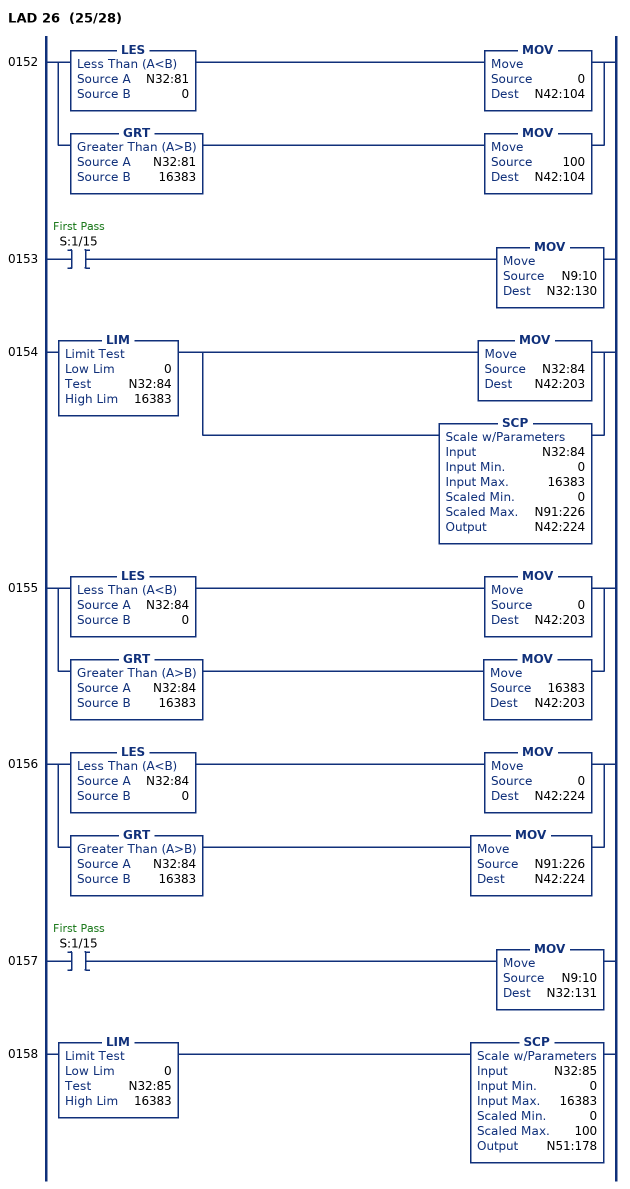
% Rung: 152 %
SOR BST LES N32:81 0 MOV 0 N42:104 NXB GRT N32:81 16383 MOV 100 N42:104 BND EOR
% Rung: 153 %
SOR XIC S:1/15 MOV N9:10 N32:130 EOR
%   S:1/15  "First Pass" %
% Rung: 154 %
SOR LIM 0 N32:84 16383 BST MOV N32:84 N42:203 NXB SCP N32:84 0 16383 0 N91:226 N42:224 BND EOR
% Rung: 155 %
SOR BST LES N32:84 0 MOV 0 N42:203 NXB GRT N32:84 16383 MOV 16383 N42:203 BND EOR
% Rung: 156 %
SOR BST LES N32:84 0 MOV 0 N42:224 NXB GRT N32:84 16383 MOV N91:226 N42:224 BND EOR
% Rung: 157 %
SOR XIC S:1/15 MOV N9:10 N32:131 EOR
%   S:1/15  "First Pass" %
% Rung: 158 %
SOR LIM 0 N32:85 16383 SCP N32:85 0 16383 0 100 N51:178 EOR

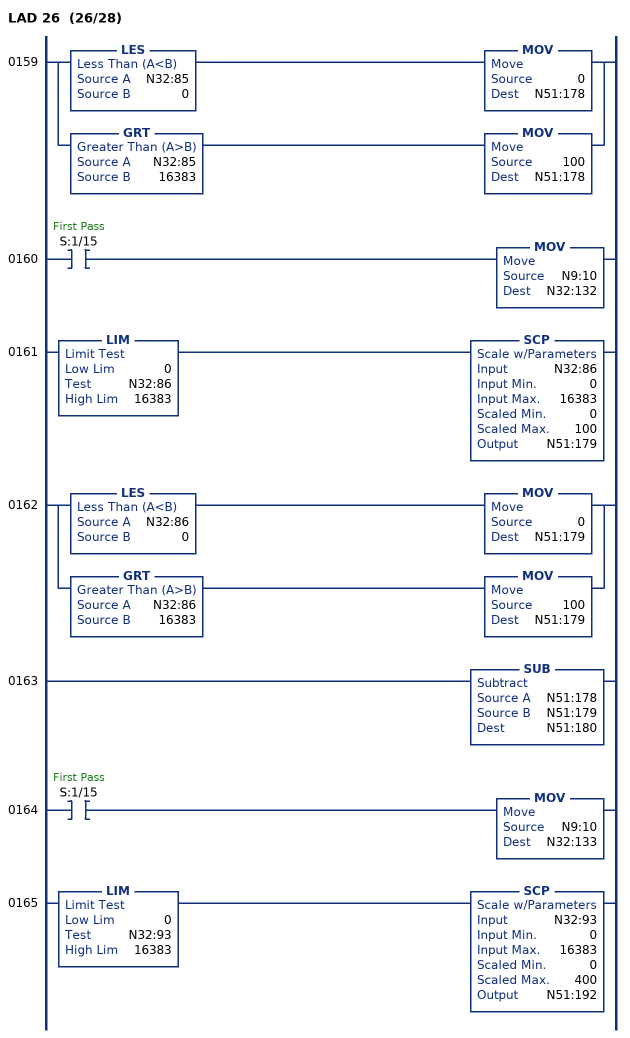
% Rung: 159 %
SOR BST LES N32:85 0 MOV 0 N51:178 NXB GRT N32:85 16383 MOV 100 N51:178 BND EOR
% Rung: 160 %
SOR XIC S:1/15 MOV N9:10 N32:132 EOR
%   S:1/15  "First Pass" %
% Rung: 161 %
SOR LIM 0 N32:86 16383 SCP N32:86 0 16383 0 100 N51:179 EOR
% Rung: 162 %
SOR BST LES N32:86 0 MOV 0 N51:179 NXB GRT N32:86 16383 MOV 100 N51:179 BND EOR
% Rung: 163 %
SOR SUB N51:178 N51:179 N51:180 EOR
% Rung: 164 %
SOR XIC S:1/15 MOV N9:10 N32:133 EOR
%   S:1/15  "First Pass" %
% Rung: 165 %
SOR LIM 0 N32:93 16383 SCP N32:93 0 16383 0 400 N51:192 EOR

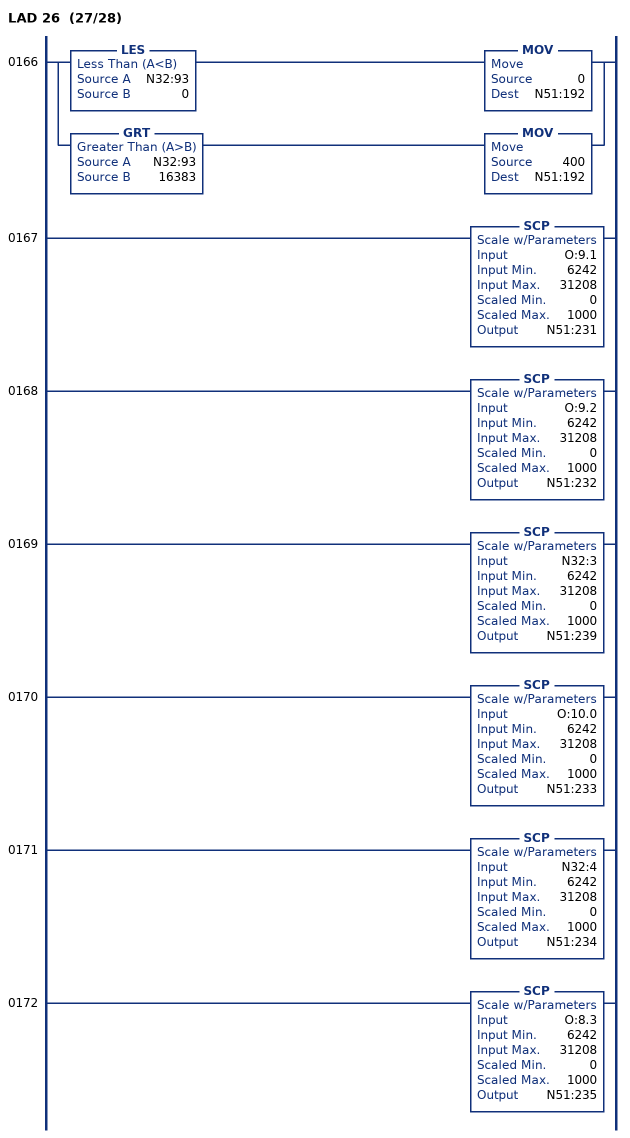
% Rung: 166 %
SOR BST LES N32:93 0 MOV 0 N51:192 NXB GRT N32:93 16383 MOV 400 N51:192 BND EOR
% Rung: 167 %
SOR SCP O:9.1 6242 31208 0 1000 N51:231 EOR
% Rung: 168 %
SOR SCP O:9.2 6242 31208 0 1000 N51:232 EOR
% Rung: 169 %
SOR SCP N32:3 6242 31208 0 1000 N51:239 EOR
% Rung: 170 %
SOR SCP O:10.0 6242 31208 0 1000 N51:233 EOR
% Rung: 171 %
SOR SCP N32:4 6242 31208 0 1000 N51:234 EOR
% Rung: 172 %
SOR SCP O:8.3 6242 31208 0 1000 N51:235 EOR

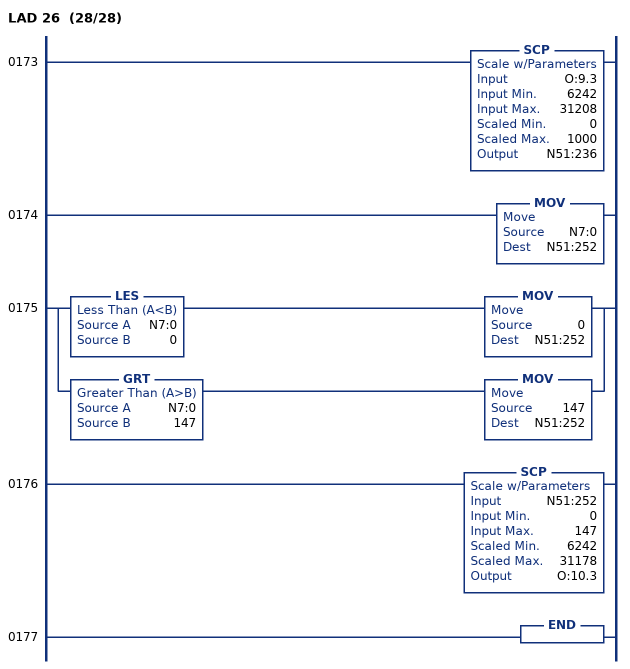
% Rung: 173 %
SOR SCP O:9.3 6242 31208 0 1000 N51:236 EOR
% Rung: 174 %
SOR MOV N7:0 N51:252 EOR
% Rung: 175 %
SOR BST LES N7:0 0 MOV 0 N51:252 NXB GRT N7:0 147 MOV 147 N51:252 BND EOR
% Rung: 176 %
SOR SCP N51:252 0 147 6242 31178 O:10.3 EOR
% Rung: 177 %
SOR END EOR

LADDER 27
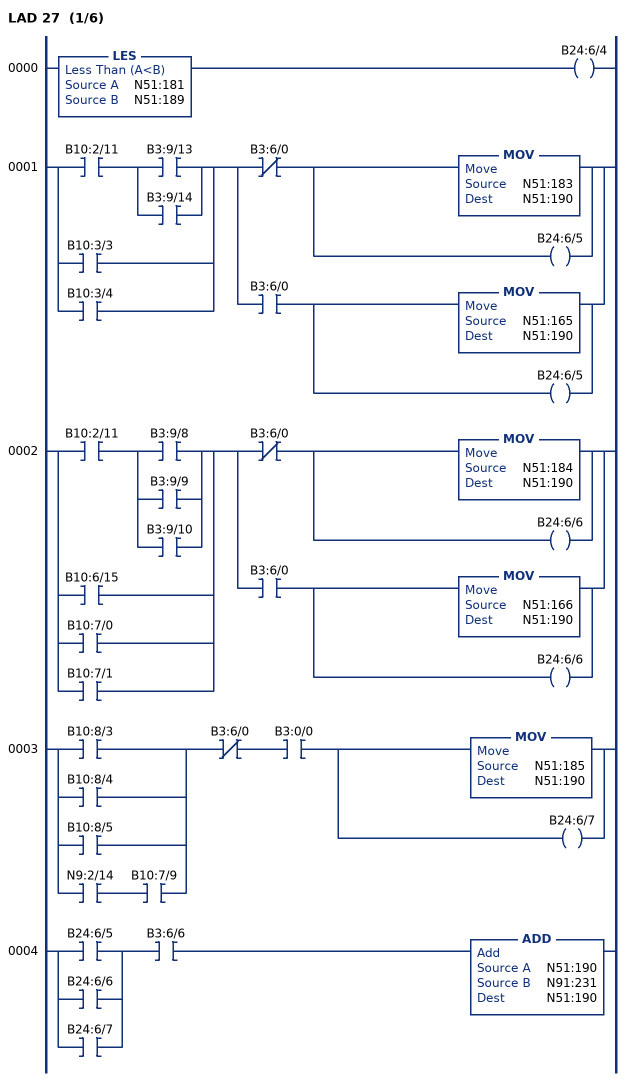
% Rung: 0 %
SOR LES N51:181 N51:189 OTE B24:6/4 EOR
% Rung: 1 %
SOR BST XIC B10:2/11 BST XIC B3:9/13 NXB XIC B3:9/14 BND NXB XIC B10:3/3 NXB XIC B10:3/4 BND BST XIO B3:6/0 BST MOV N51:183 N51:190 NXB OTE B24:6/5 BND NXB XIC B3:6/0 BST MOV N51:165 N51:190 NXB OTE B24:6/5 BND BND EOR
% Rung: 2 %
SOR BST XIC B10:2/11 BST XIC B3:9/8 NXB XIC B3:9/9 NXB XIC B3:9/10 BND NXB XIC B10:6/15 NXB XIC B10:7/0 NXB XIC B10:7/1 BND BST XIO B3:6/0 BST MOV N51:184 N51:190 NXB OTE B24:6/6 BND NXB XIC B3:6/0 BST MOV N51:166 N51:190 NXB OTE B24:6/6 BND BND EOR
% Rung: 3 %
SOR BST XIC B10:8/3 NXB XIC B10:8/4 NXB XIC B10:8/5 NXB XIC N9:2/14 XIC B10:7/9 BND XIO B3:6/0 XIC B3:0/0 BST MOV N51:185 N51:190 NXB OTE B24:6/7 BND EOR
% Rung: 4 %
SOR BST XIC B24:6/5 NXB XIC B24:6/6 NXB XIC B24:6/7 BND XIC B3:6/6 ADD N51:190 N91:231 N51:190 EOR

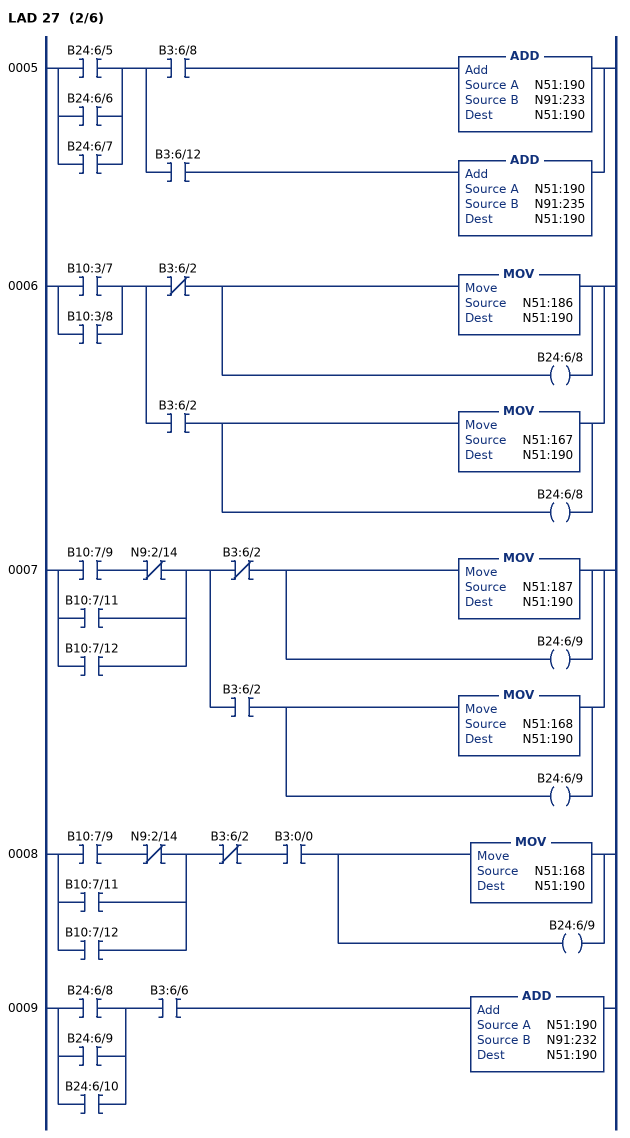
% Rung: 5 %
SOR BST XIC B24:6/5 NXB XIC B24:6/6 NXB XIC B24:6/7 BND BST XIC B3:6/8 ADD N51:190 N91:233 N51:190 NXB XIC B3:6/12 ADD N51:190 N91:235 N51:190 BND EOR
% Rung: 6 %
SOR BST XIC B10:3/7 NXB XIC B10:3/8 BND BST XIO B3:6/2 BST MOV N51:186 N51:190 NXB OTE B24:6/8 BND NXB XIC B3:6/2 BST MOV N51:167 N51:190 NXB OTE B24:6/8 BND BND EOR
% Rung: 7 %
SOR BST XIC B10:7/9 XIO N9:2/14 NXB XIC B10:7/11 NXB XIC B10:7/12 BND BST XIO B3:6/2 BST MOV N51:187 N51:190 NXB OTE B24:6/9 BND NXB XIC B3:6/2 BST MOV N51:168 N51:190 NXB OTE B24:6/9 BND BND EOR
% Rung: 8 %
SOR BST XIC B10:7/9 XIO N9:2/14 NXB XIC B10:7/11 NXB XIC B10:7/12 BND XIO B3:6/2 XIC B3:0/0 BST MOV N51:168 N51:190 NXB OTE B24:6/9 BND EOR
% Rung: 9 %
SOR BST XIC B24:6/8 NXB XIC B24:6/9 NXB XIC B24:6/10 BND XIC B3:6/6 ADD N51:190 N91:232 N51:190 EOR

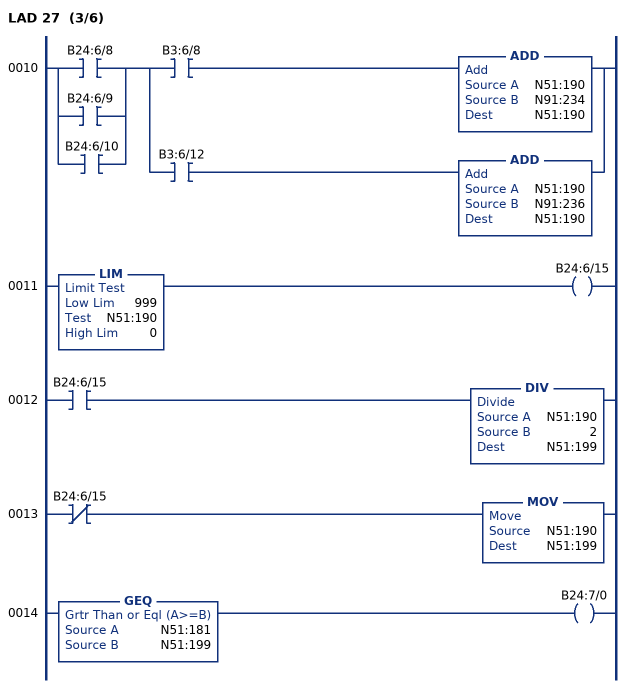
% Rung: 10 %
SOR BST XIC B24:6/8 NXB XIC B24:6/9 NXB XIC B24:6/10 BND BST XIC B3:6/8 ADD N51:190 N91:234 N51:190 NXB XIC B3:6/12 ADD N51:190 N91:236 N51:190 BND EOR
% Rung: 11 %
SOR LIM 999 N51:190 0 OTE B24:6/15 EOR
% Rung: 12 %
SOR XIC B24:6/15 DIV N51:190 2 N51:199 EOR
% Rung: 13 %
SOR XIO B24:6/15 MOV N51:190 N51:199 EOR
% Rung: 14 %
SOR GEQ N51:181 N51:199 OTE B24:7/0 EOR

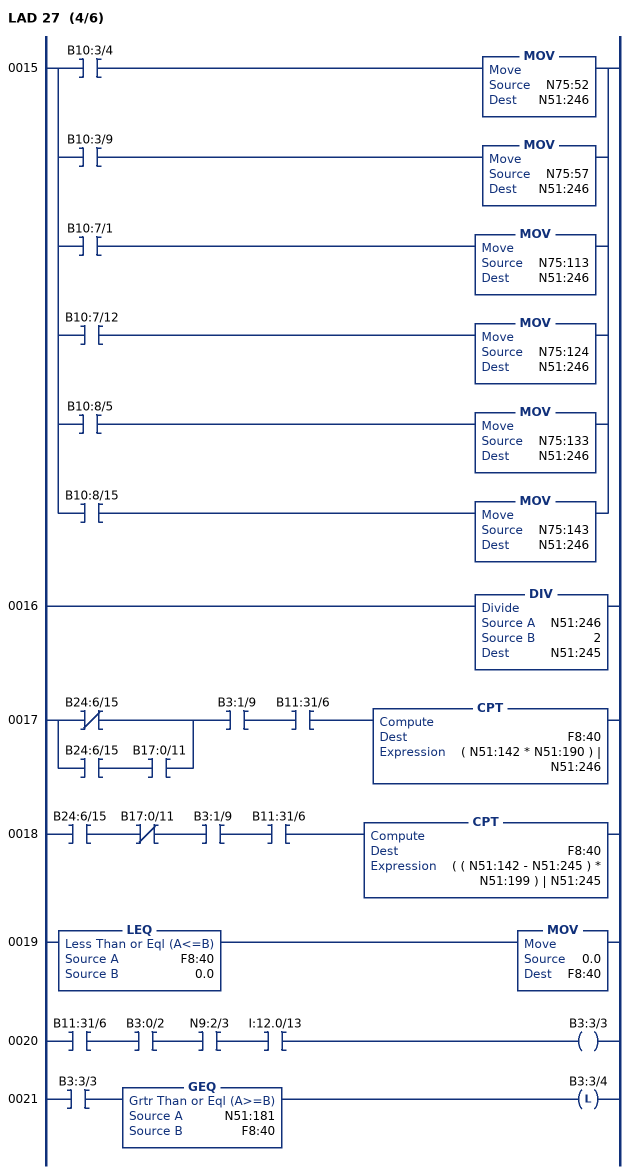
% Rung: 15 %
SOR BST XIC B10:3/4 MOV N75:52 N51:246 NXB XIC B10:3/9 MOV N75:57 N51:246 NXB XIC B10:7/1 MOV N75:113 N51:246 NXB XIC B10:7/12 MOV N75:124 N51:246 NXB XIC B10:8/5 MOV N75:133 N51:246 NXB XIC B10:8/15 MOV N75:143 N51:246 BND EOR
% Rung: 16 %
SOR DIV N51:246 2 N51:245 EOR
% Rung: 17 %
SOR BST XIO B24:6/15 NXB XIC B24:6/15 XIC B17:0/11 BND XIC B3:1/9 XIC B11:31/6 CPT F8:40 " ( N51:142 * N51:190 ) | N51:246 " EOR
% Rung: 18 %
SOR XIC B24:6/15 XIO B17:0/11 XIC B3:1/9 XIC B11:31/6 CPT F8:40 " ( ( N51:142 - N51:245 ) * N51:199 ) | N51:245 " EOR
% Rung: 19 %
SOR LEQ F8:40 0.0 MOV 0.0 F8:40 EOR
% Rung: 20 %
SOR XIC B11:31/6 XIC B3:0/2 XIC N9:2/3 XIC I:12.0/13 OTE B3:3/3 EOR
% Rung: 21 %
SOR XIC B3:3/3 GEQ N51:181 F8:40 OTL B3:3/4 EOR

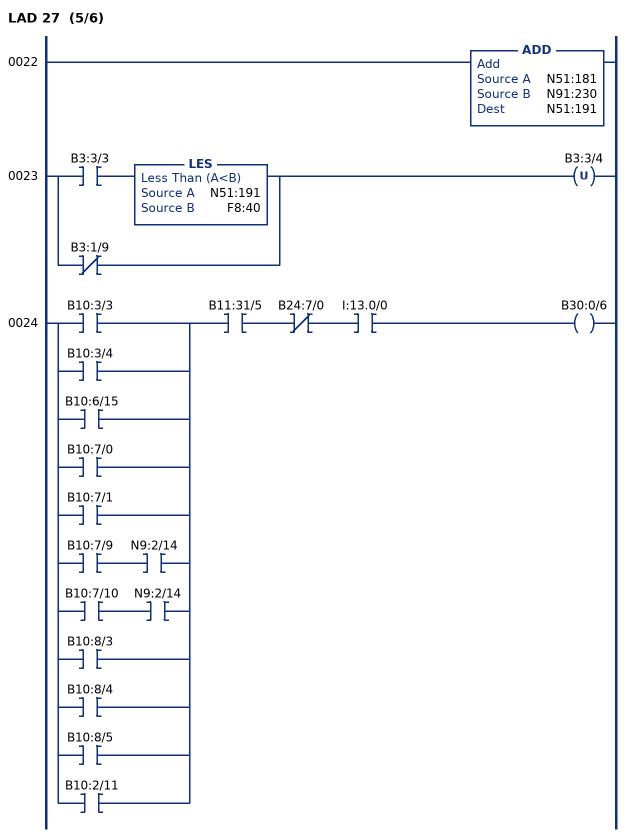
% Rung: 22 %
SOR ADD N51:181 N91:230 N51:191 EOR
% Rung: 23 %
SOR BST XIC B3:3/3 LES N51:191 F8:40 NXB XIO B3:1/9 BND OTU B3:3/4 EOR
% Rung: 24 %
SOR BST XIC B10:3/3 NXB XIC B10:3/4 NXB XIC B10:6/15 NXB XIC B10:7/0 NXB XIC B10:7/1 NXB XIC B10:7/9 XIC N9:2/14 NXB XIC B10:7/10 XIC N9:2/14 NXB XIC B10:8/3 NXB XIC B10:8/4 NXB XIC B10:8/5 NXB XIC B10:2/11 BND XIC B11:31/5 XIO B24:7/0 XIC I:13.0/0 OTE B30:0/6 EOR

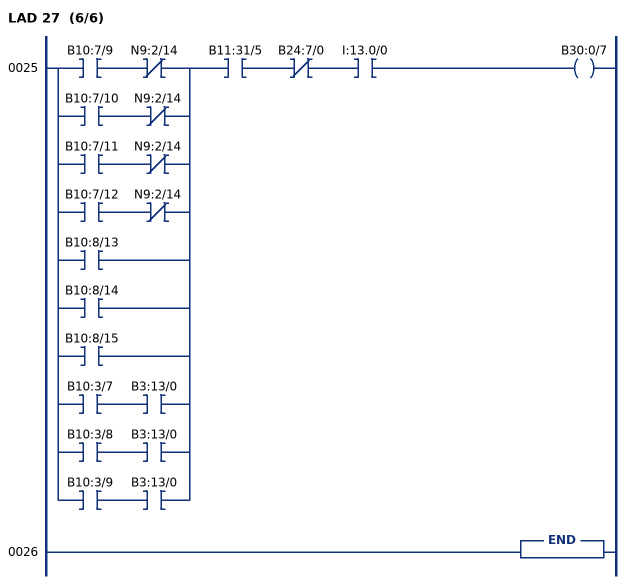
% Rung: 25 %
SOR BST XIC B10:7/9 XIO N9:2/14 NXB XIC B10:7/10 XIO N9:2/14 NXB XIC B10:7/11 XIO N9:2/14 NXB XIC B10:7/12 XIO N9:2/14 NXB XIC B10:8/13 NXB XIC B10:8/14 NXB XIC B10:8/15 NXB XIC B10:3/7 XIC B3:13/0 NXB XIC B10:3/8 XIC B3:13/0 NXB XIC B10:3/9 XIC B3:13/0 BND XIC B11:31/5 XIO B24:7/0 XIC I:13.0/0 OTE B30:0/7 EOR
% Rung: 26 %
SOR END EOR

LADDER 28
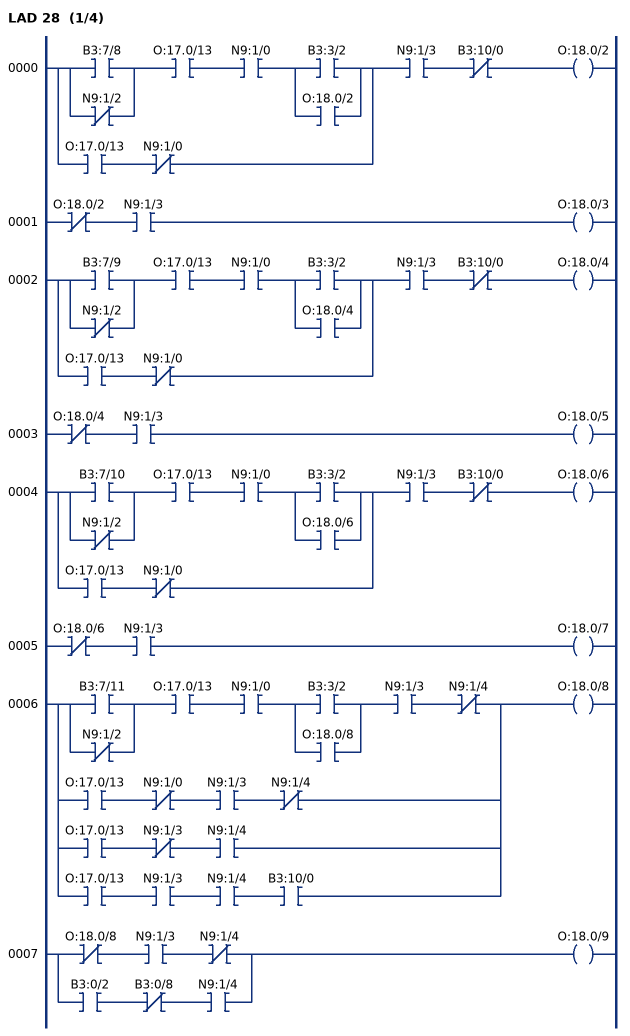
% Rung: 0 %
SOR BST BST XIC B3:7/8 NXB XIO N9:1/2 BND XIC O:17.0/13 XIC N9:1/0 BST XIC B3:3/2 NXB XIC O:18.0/2 BND NXB XIC O:17.0/13 XIO N9:1/0 BND XIC N9:1/3 XIO B3:10/0 OTE O:18.0/2 EOR
% Rung: 1 %
SOR XIO O:18.0/2 XIC N9:1/3 OTE O:18.0/3 EOR
% Rung: 2 %
SOR BST BST XIC B3:7/9 NXB XIO N9:1/2 BND XIC O:17.0/13 XIC N9:1/0 BST XIC B3:3/2 NXB XIC O:18.0/4 BND NXB XIC O:17.0/13 XIO N9:1/0 BND XIC N9:1/3 XIO B3:10/0 OTE O:18.0/4 EOR
% Rung: 3 %
SOR XIO O:18.0/4 XIC N9:1/3 OTE O:18.0/5 EOR
% Rung: 4 %
SOR BST BST XIC B3:7/10 NXB XIO N9:1/2 BND XIC O:17.0/13 XIC N9:1/0 BST XIC B3:3/2 NXB XIC O:18.0/6 BND NXB XIC O:17.0/13 XIO N9:1/0 BND XIC N9:1/3 XIO B3:10/0 OTE O:18.0/6 EOR
% Rung: 5 %
SOR XIO O:18.0/6 XIC N9:1/3 OTE O:18.0/7 EOR
% Rung: 6 %
SOR BST BST XIC B3:7/11 NXB XIO N9:1/2 BND XIC O:17.0/13 XIC N9:1/0 BST XIC B3:3/2 NXB XIC O:18.0/8 BND XIC N9:1/3 XIO N9:1/4 NXB XIC O:17.0/13 XIO N9:1/0 XIC N9:1/3 XIO N9:1/4 NXB XIC O:17.0/13 XIO N9:1/3 XIC N9:1/4 NXB XIC O:17.0/13 XIC N9:1/3 XIC N9:1/4 XIC B3:10/0 BND OTE O:18.0/8 EOR
% Rung: 7 %
SOR BST XIO O:18.0/8 XIC N9:1/3 XIO N9:1/4 NXB XIC B3:0/2 XIO B3:0/8 XIC N9:1/4 BND OTE O:18.0/9 EOR

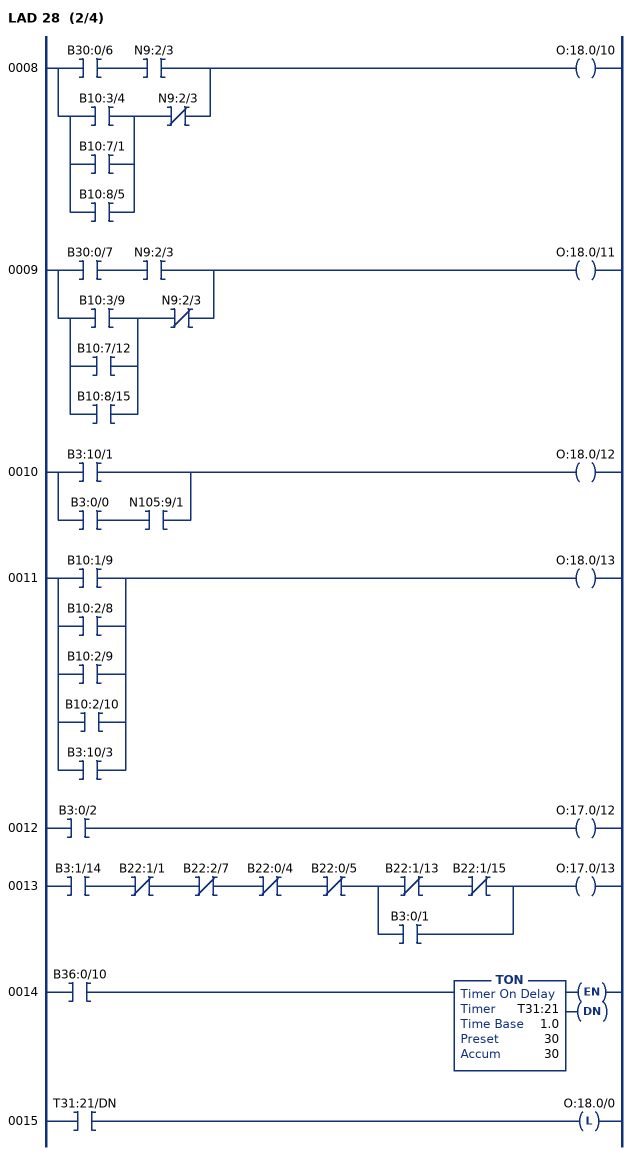
% Rung: 8 %
SOR BST XIC B30:0/6 XIC N9:2/3 NXB BST XIC B10:3/4 NXB XIC B10:7/1 NXB XIC B10:8/5 BND XIO N9:2/3 BND OTE O:18.0/10 EOR
% Rung: 9 %
SOR BST XIC B30:0/7 XIC N9:2/3 NXB BST XIC B10:3/9 NXB XIC B10:7/12 NXB XIC B10:8/15 BND XIO N9:2/3 BND OTE O:18.0/11 EOR
% Rung: 10 %
SOR BST XIC B3:10/1 NXB XIC B3:0/0 XIC N105:9/1 BND OTE O:18.0/12 EOR
% Rung: 11 %
SOR BST XIC B10:1/9 NXB XIC B10:2/8 NXB XIC B10:2/9 NXB XIC B10:2/10 NXB XIC B3:10/3 BND OTE O:18.0/13 EOR
% Rung: 12 %
SOR XIC B3:0/2 OTE O:17.0/12 EOR
% Rung: 13 %
SOR XIC B3:1/14 XIO B22:1/1 XIO B22:2/7 XIO B22:0/4 XIO B22:0/5 BST XIO B22:1/13 XIO B22:1/15 NXB XIC B3:0/1 BND OTE O:17.0/13 EOR
% Rung: 14 %
SOR XIC B36:0/10 TON T31:21 1.0 30 30 EOR
% Rung: 15 %
SOR XIC T31:21/DN OTL O:18.0/0 EOR

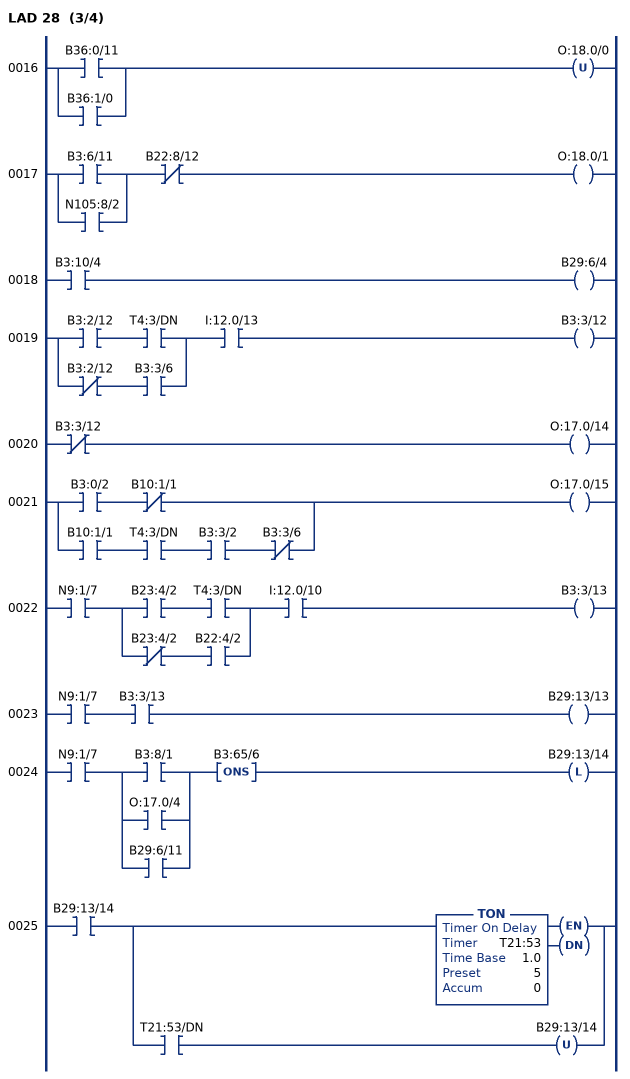
% Rung: 16 %
SOR BST XIC B36:0/11 NXB XIC B36:1/0 BND OTU O:18.0/0 EOR
% Rung: 17 %
SOR BST XIC B3:6/11 NXB XIC N105:8/2 BND XIO B22:8/12 OTE O:18.0/1 EOR
% Rung: 18 %
SOR XIC B3:10/4 OTE B29:6/4 EOR
% Rung: 19 %
SOR BST XIC B3:2/12 XIC T4:3/DN NXB XIO B3:2/12 XIC B3:3/6 BND XIC I:12.0/13 OTE B3:3/12 EOR
% Rung: 20 %
SOR XIO B3:3/12 OTE O:17.0/14 EOR
% Rung: 21 %
SOR BST XIC B3:0/2 XIO B10:1/1 NXB XIC B10:1/1 XIC T4:3/DN XIC B3:3/2 XIO B3:3/6 BND OTE O:17.0/15 EOR
% Rung: 22 %
SOR XIC N9:1/7 BST XIC B23:4/2 XIC T4:3/DN NXB XIO B23:4/2 XIC B22:4/2 BND XIC I:12.0/10 OTE B3:3/13 EOR
% Rung: 23 %
SOR XIC N9:1/7 XIC B3:3/13 OTE B29:13/13 EOR
% Rung: 24 %
SOR XIC N9:1/7 BST XIC B3:8/1 NXB XIC O:17.0/4 NXB XIC B29:6/11 BND OSR B3:65/6 OTL B29:13/14 EOR
% Rung: 25 %
SOR XIC B29:13/14 BST TON T21:53 1.0 5 0 NXB XIC T21:53/DN OTU B29:13/14 BND EOR

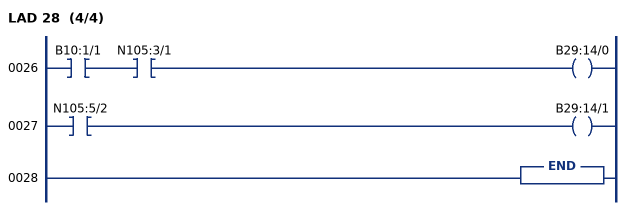
% Rung: 26 %
SOR XIC B10:1/1 XIC N105:3/1 OTE B29:14/0 EOR
% Rung: 27 %
SOR XIC N105:5/2 OTE B29:14/1 EOR
% Rung: 28 %
SOR END EOR

LADDER 31
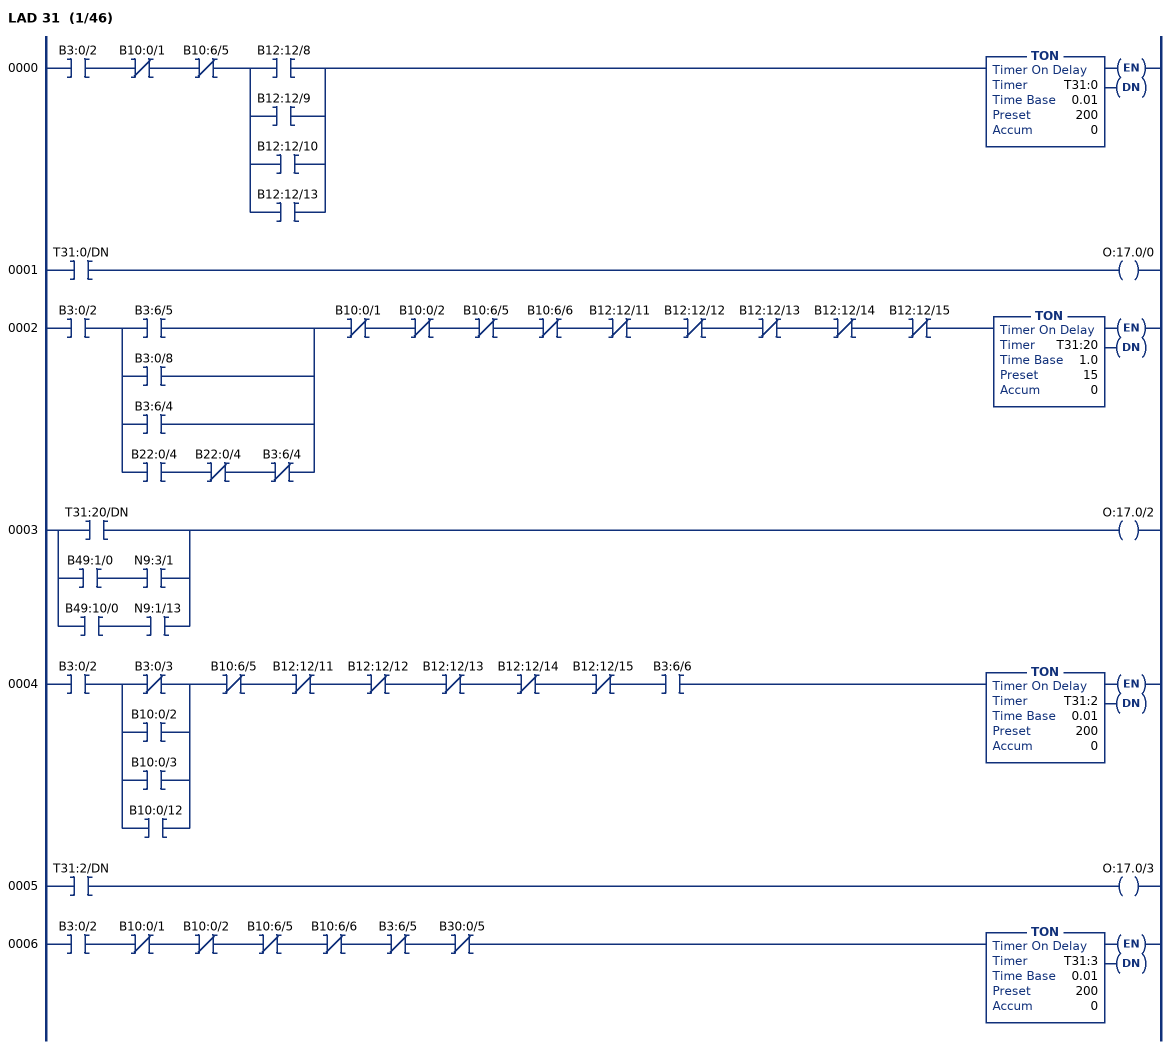
% Rung: 0 %
SOR XIC B3:0/2 XIO B10:0/1 XIO B10:6/5 BST XIC B12:12/8 NXB XIC B12:12/9 NXB XIC B12:12/10 NXB XIC B12:12/13 BND TON T31:0 0.01 200 0 EOR
% Rung: 1 %
SOR XIC T31:0/DN OTE O:17.0/0 EOR
% Rung: 2 %
SOR XIC B3:0/2 BST XIC B3:6/5 NXB XIC B3:0/8 NXB XIC B3:6/4 NXB XIC B22:0/4 XIO B22:0/4 XIO B3:6/4 BND XIO B10:0/1 XIO B10:0/2 XIO B10:6/5 XIO B10:6/6 XIO B12:12/11 XIO B12:12/12 XIO B12:12/13 XIO B12:12/14 XIO B12:12/15 TON T31:20 1.0 15 0 EOR
% Rung: 3 %
SOR BST XIC T31:20/DN NXB XIC B49:1/0 XIC N9:3/1 NXB XIC B49:10/0 XIC N9:1/13 BND OTE O:17.0/2 EOR
% Rung: 4 %
SOR XIC B3:0/2 BST XIO B3:0/3 NXB XIC B10:0/2 NXB XIC B10:0/3 NXB XIC B10:0/12 BND XIO B10:6/5 XIO B12:12/11 XIO B12:12/12 XIO B12:12/13 XIO B12:12/14 XIO B12:12/15 XIC B3:6/6 TON T31:2 0.01 200 0 EOR
% Rung: 5 %
SOR XIC T31:2/DN OTE O:17.0/3 EOR
% Rung: 6 %
SOR XIC B3:0/2 XIO B10:0/1 XIO B10:0/2 XIO B10:6/5 XIO B10:6/6 XIO B3:6/5 XIO B30:0/5 TON T31:3 0.01 200 0 EOR

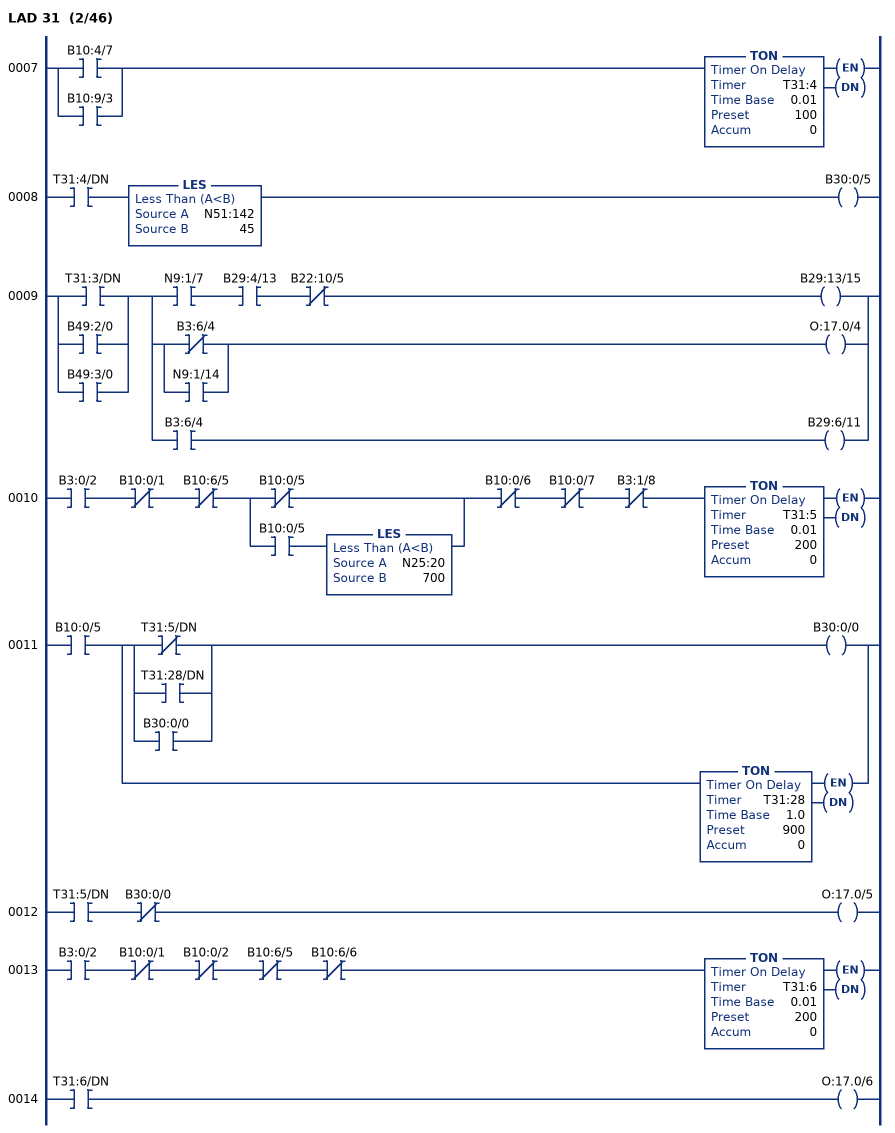
% Rung: 7 %
SOR BST XIC B10:4/7 NXB XIC B10:9/3 BND TON T31:4 0.01 100 0 EOR
% Rung: 8 %
SOR XIC T31:4/DN LES N51:142 45 OTE B30:0/5 EOR
% Rung: 9 %
SOR BST XIC T31:3/DN NXB XIC B49:2/0 NXB XIC B49:3/0 BND BST XIC N9:1/7 XIC B29:4/13 XIO B22:10/5 OTE B29:13/15 NXB BST XIO B3:6/4 NXB XIC N9:1/14 BND OTE O:17.0/4 NXB XIC B3:6/4 OTE B29:6/11 BND EOR
% Rung: 10 %
SOR XIC B3:0/2 XIO B10:0/1 XIO B10:6/5 BST XIO B10:0/5 NXB XIC B10:0/5 LES N25:20 700 BND XIO B10:0/6 XIO B10:0/7 XIO B3:1/8 TON T31:5 0.01 200 0 EOR
% Rung: 11 %
SOR XIC B10:0/5 BST BST XIO T31:5/DN NXB XIC T31:28/DN NXB XIC B30:0/0 BND OTE B30:0/0 NXB TON T31:28 1.0 900 0 BND EOR
% Rung: 12 %
SOR XIC T31:5/DN XIO B30:0/0 OTE O:17.0/5 EOR
% Rung: 13 %
SOR XIC B3:0/2 XIO B10:0/1 XIO B10:0/2 XIO B10:6/5 XIO B10:6/6 TON T31:6 0.01 200 0 EOR
% Rung: 14 %
SOR XIC T31:6/DN OTE O:17.0/6 EOR

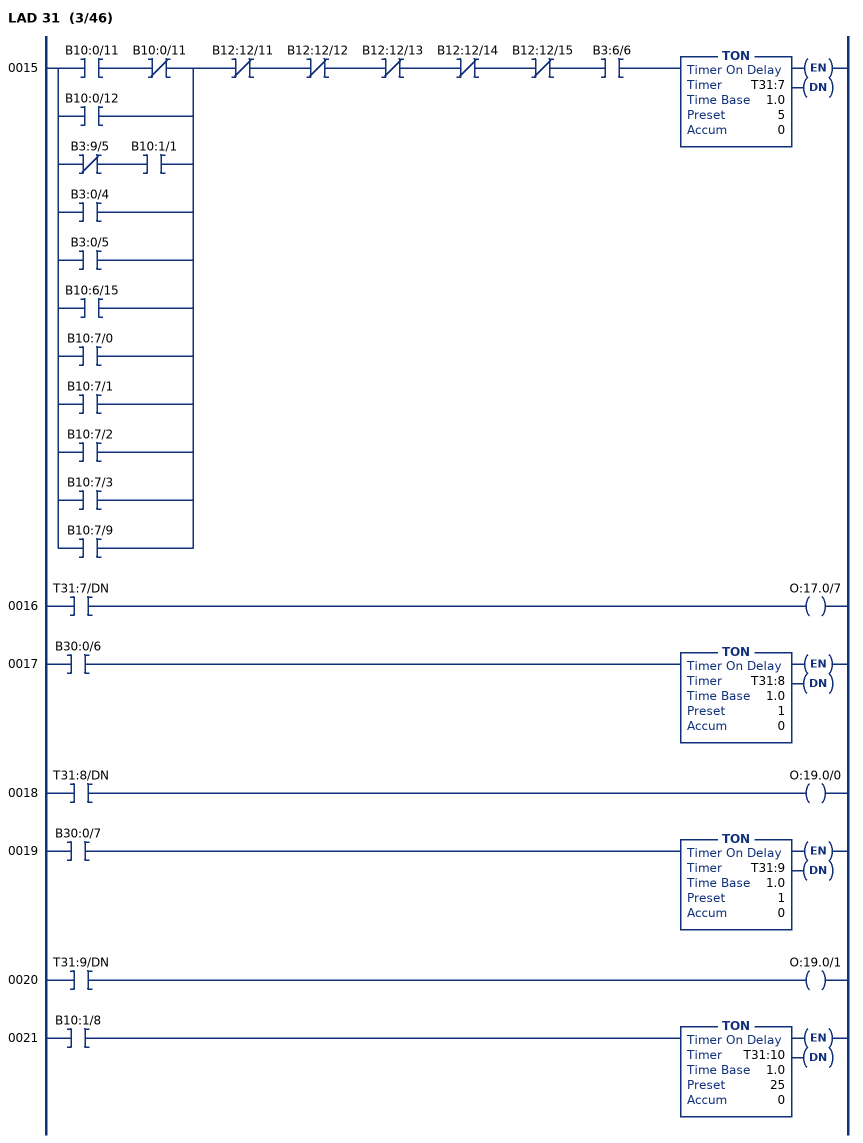
% Rung: 15 %
SOR BST XIC B10:0/11 XIO B10:0/11 NXB XIC B10:0/12 NXB XIO B3:9/5 XIC B10:1/1 NXB XIC B3:0/4 NXB XIC B3:0/5 NXB XIC B10:6/15 NXB XIC B10:7/0 NXB XIC B10:7/1 NXB XIC B10:7/2 NXB XIC B10:7/3 NXB XIC B10:7/9 BND XIO B12:12/11 XIO B12:12/12 XIO B12:12/13 XIO B12:12/14 XIO B12:12/15 XIC B3:6/6 TON T31:7 1.0 5 0 EOR
% Rung: 16 %
SOR XIC T31:7/DN OTE O:17.0/7 EOR
% Rung: 17 %
SOR XIC B30:0/6 TON T31:8 1.0 1 0 EOR
% Rung: 18 %
SOR XIC T31:8/DN OTE O:19.0/0 EOR
% Rung: 19 %
SOR XIC B30:0/7 TON T31:9 1.0 1 0 EOR
% Rung: 20 %
SOR XIC T31:9/DN OTE O:19.0/1 EOR
% Rung: 21 %
SOR XIC B10:1/8 TON T31:10 1.0 25 0 EOR

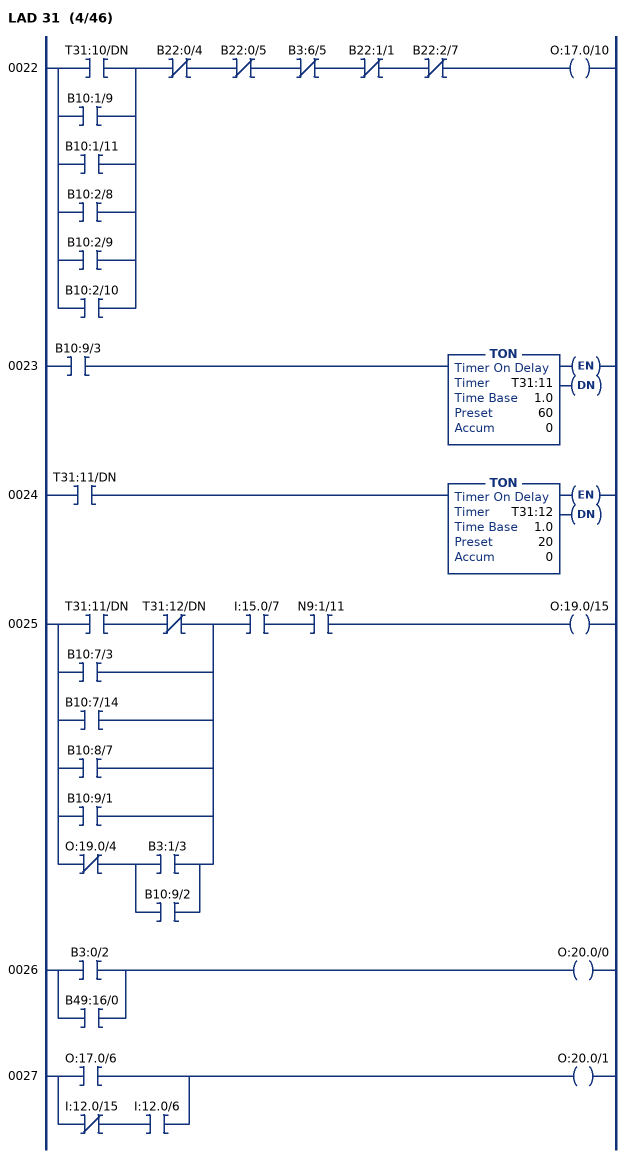
% Rung: 22 %
SOR BST XIC T31:10/DN NXB XIC B10:1/9 NXB XIC B10:1/11 NXB XIC B10:2/8 NXB XIC B10:2/9 NXB XIC B10:2/10 BND XIO B22:0/4 XIO B22:0/5 XIO B3:6/5 XIO B22:1/1 XIO B22:2/7 OTE O:17.0/10 EOR
% Rung: 23 %
SOR XIC B10:9/3 TON T31:11 1.0 60 0 EOR
% Rung: 24 %
SOR XIC T31:11/DN TON T31:12 1.0 20 0 EOR
% Rung: 25 %
SOR BST XIC T31:11/DN XIO T31:12/DN NXB XIC B10:7/3 NXB XIC B10:7/14 NXB XIC B10:8/7 NXB XIC B10:9/1 NXB XIO O:19.0/4 BST XIC B3:1/3 NXB XIC B10:9/2 BND BND XIC I:15.0/7 XIC N9:1/11 OTE O:19.0/15 EOR
% Rung: 26 %
SOR BST XIC B3:0/2 NXB XIC B49:16/0 BND OTE O:20.0/0 EOR
% Rung: 27 %
SOR BST XIC O:17.0/6 NXB XIO I:12.0/15 XIC I:12.0/6 BND OTE O:20.0/1 EOR

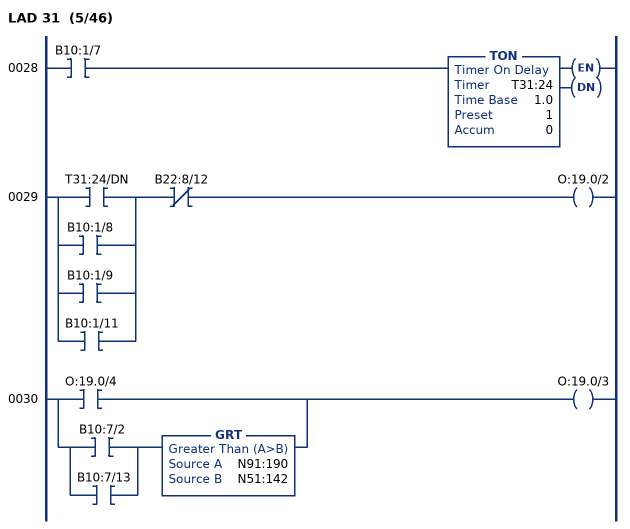
% Rung: 28 %
SOR XIC B10:1/7 TON T31:24 1.0 1 0 EOR
% Rung: 29 %
SOR BST XIC T31:24/DN NXB XIC B10:1/8 NXB XIC B10:1/9 NXB XIC B10:1/11 BND XIO B22:8/12 OTE O:19.0/2 EOR
% Rung: 30 %
SOR BST XIC O:19.0/4 NXB BST XIC B10:7/2 NXB XIC B10:7/13 BND GRT N91:190 N51:142 BND OTE O:19.0/3 EOR

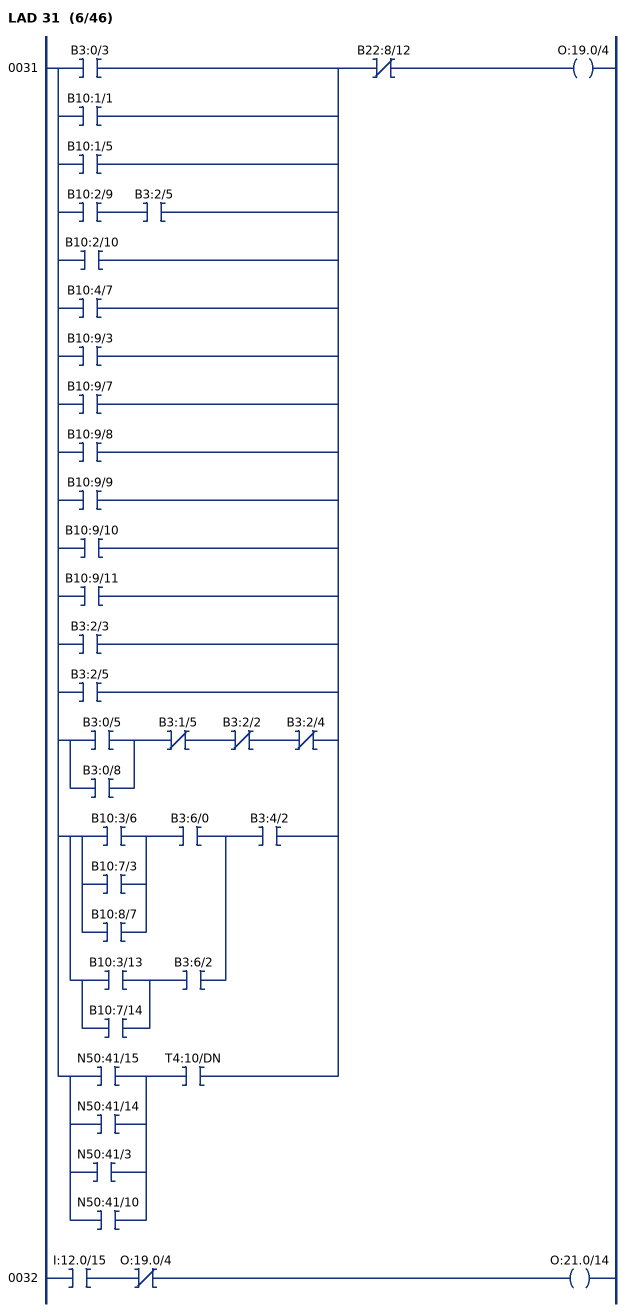
% Rung: 31 %
SOR BST XIC B3:0/3 NXB XIC B10:1/1 NXB XIC B10:1/5 NXB XIC B10:2/9 XIC B3:2/5 NXB XIC B10:2/10 NXB XIC B10:4/7 NXB XIC B10:9/3 NXB XIC B10:9/7 NXB XIC B10:9/8 NXB XIC B10:9/9 NXB XIC B10:9/10 NXB XIC B10:9/11 NXB XIC B3:2/3 NXB XIC B3:2/5 NXB BST XIC B3:0/5 NXB XIC B3:0/8 BND XIO B3:1/5 XIO B3:2/2 XIO B3:2/4 NXB BST BST XIC B10:3/6 NXB XIC B10:7/3 NXB XIC B10:8/7 BND XIC B3:6/0 NXB BST XIC B10:3/13 NXB XIC B10:7/14 BND XIC B3:6/2 BND XIC B3:4/2 NXB BST XIC N50:41/15 NXB XIC N50:41/14 NXB XIC N50:41/3 NXB XIC N50:41/10 BND XIC T4:10/DN BND XIO B22:8/12 OTE O:19.0/4 EOR
% Rung: 32 %
SOR XIC I:12.0/15 XIO O:19.0/4 OTE O:21.0/14 EOR

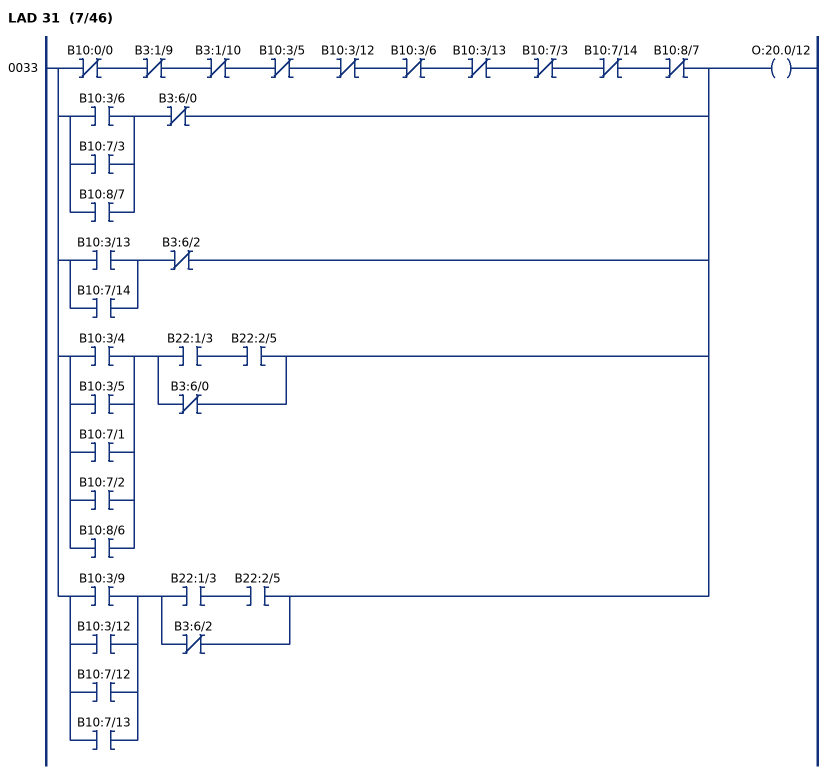
% Rung: 33 %
SOR BST XIO B10:0/0 XIO B3:1/9 XIO B3:1/10 XIO B10:3/5 XIO B10:3/12 XIO B10:3/6 XIO B10:3/13 XIO B10:7/3 XIO B10:7/14 XIO B10:8/7 NXB BST XIC B10:3/6 NXB XIC B10:7/3 NXB XIC B10:8/7 BND XIO B3:6/0 NXB BST XIC B10:3/13 NXB XIC B10:7/14 BND XIO B3:6/2 NXB BST XIC B10:3/4 NXB XIC B10:3/5 NXB XIC B10:7/1 NXB XIC B10:7/2 NXB XIC B10:8/6 BND BST XIC B22:1/3 XIC B22:2/5 NXB XIO B3:6/0 BND NXB BST XIC B10:3/9 NXB XIC B10:3/12 NXB XIC B10:7/12 NXB XIC B10:7/13 BND BST XIC B22:1/3 XIC B22:2/5 NXB XIO B3:6/2 BND BND OTE O:20.0/12 EOR

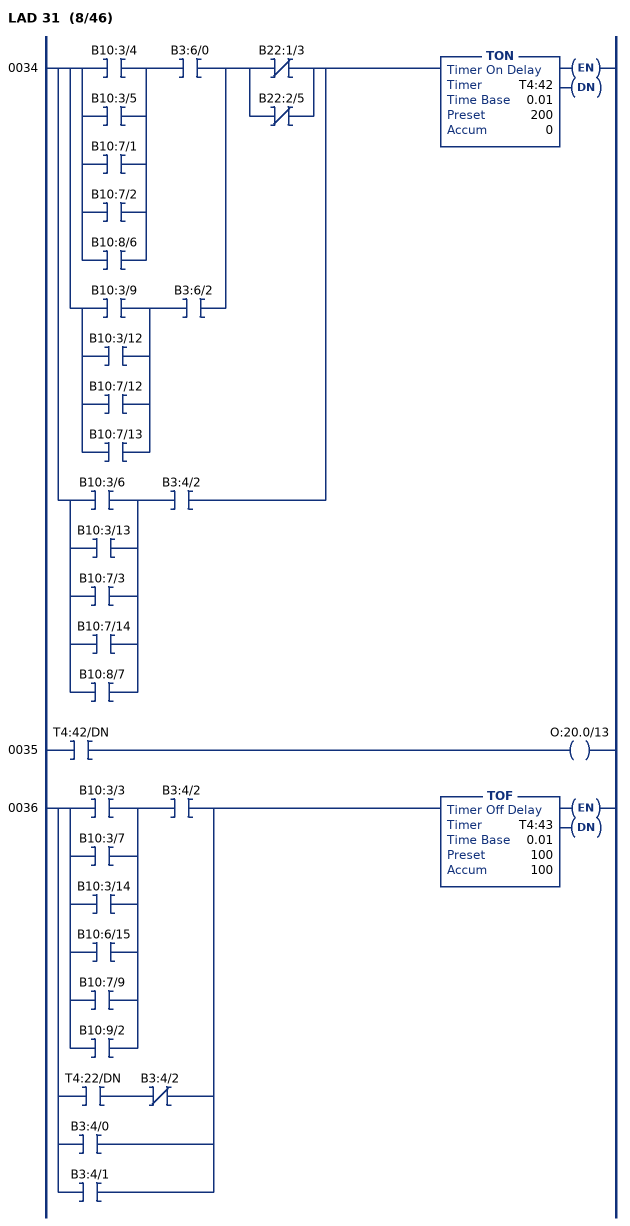
% Rung: 34 %
SOR BST BST BST XIC B10:3/4 NXB XIC B10:3/5 NXB XIC B10:7/1 NXB XIC B10:7/2 NXB XIC B10:8/6 BND XIC B3:6/0 NXB BST XIC B10:3/9 NXB XIC B10:3/12 NXB XIC B10:7/12 NXB XIC B10:7/13 BND XIC B3:6/2 BND BST XIO B22:1/3 NXB XIO B22:2/5 BND NXB BST XIC B10:3/6 NXB XIC B10:3/13 NXB XIC B10:7/3 NXB XIC B10:7/14 NXB XIC B10:8/7 BND XIC B3:4/2 BND TON T4:42 0.01 200 0 EOR
% Rung: 35 %
SOR XIC T4:42/DN OTE O:20.0/13 EOR
% Rung: 36 %
SOR BST BST XIC B10:3/3 NXB XIC B10:3/7 NXB XIC B10:3/14 NXB XIC B10:6/15 NXB XIC B10:7/9 NXB XIC B10:9/2 BND XIC B3:4/2 NXB XIC T4:22/DN XIO B3:4/2 NXB XIC B3:4/0 NXB XIC B3:4/1 BND TOF T4:43 0.01 100 100 EOR

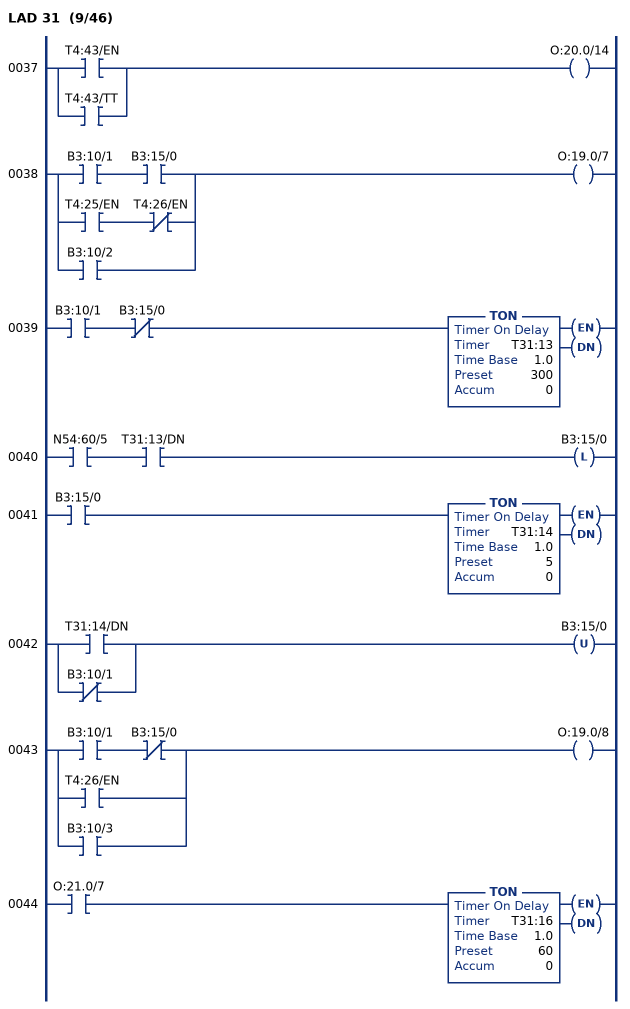
% Rung: 37 %
SOR BST XIC T4:43/EN NXB XIC T4:43/TT BND OTE O:20.0/14 EOR
% Rung: 38 %
SOR BST XIC B3:10/1 XIC B3:15/0 NXB XIC T4:25/EN XIO T4:26/EN NXB XIC B3:10/2 BND OTE O:19.0/7 EOR
% Rung: 39 %
SOR XIC B3:10/1 XIO B3:15/0 TON T31:13 1.0 300 0 EOR
% Rung: 40 %
SOR XIC N54:60/5 XIC T31:13/DN OTL B3:15/0 EOR
% Rung: 41 %
SOR XIC B3:15/0 TON T31:14 1.0 5 0 EOR
% Rung: 42 %
SOR BST XIC T31:14/DN NXB XIO B3:10/1 BND OTU B3:15/0 EOR
% Rung: 43 %
SOR BST XIC B3:10/1 XIO B3:15/0 NXB XIC T4:26/EN NXB XIC B3:10/3 BND OTE O:19.0/8 EOR
% Rung: 44 %
SOR XIC O:21.0/7 TON T31:16 1.0 60 0 EOR

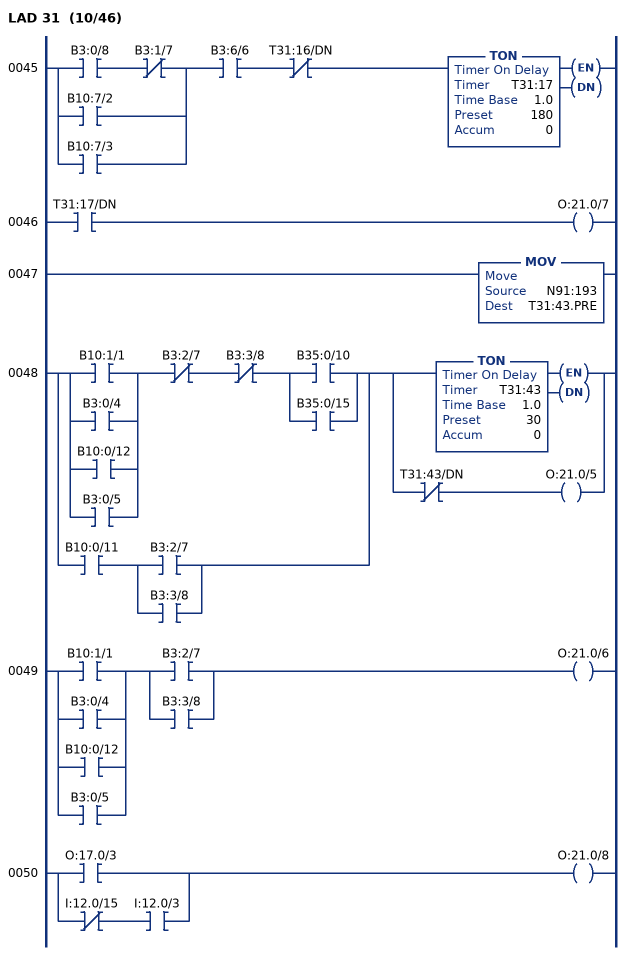
% Rung: 45 %
SOR BST XIC B3:0/8 XIO B3:1/7 NXB XIC B10:7/2 NXB XIC B10:7/3 BND XIC B3:6/6 XIO T31:16/DN TON T31:17 1.0 180 0 EOR
% Rung: 46 %
SOR XIC T31:17/DN OTE O:21.0/7 EOR
% Rung: 47 %
SOR MOV N91:193 T31:43.PRE EOR
% Rung: 48 %
SOR BST BST XIC B10:1/1 NXB XIC B3:0/4 NXB XIC B10:0/12 NXB XIC B3:0/5 BND XIO B3:2/7 XIO B3:3/8 BST XIC B35:0/10 NXB XIC B35:0/15 BND NXB XIC B10:0/11 BST XIC B3:2/7 NXB XIC B3:3/8 BND BND BST TON T31:43 1.0 30 0 NXB XIO T31:43/DN OTE O:21.0/5 BND EOR
% Rung: 49 %
SOR BST XIC B10:1/1 NXB XIC B3:0/4 NXB XIC B10:0/12 NXB XIC B3:0/5 BND BST XIC B3:2/7 NXB XIC B3:3/8 BND OTE O:21.0/6 EOR
% Rung: 50 %
SOR BST XIC O:17.0/3 NXB XIO I:12.0/15 XIC I:12.0/3 BND OTE O:21.0/8 EOR

